{attribute addProperty BoxType "KL6224-0001"}
{attribute addProperty Id "Channel_1Channel_BED7D40000"}
{attribute addProperty CRC "1796210049"}
{attribute addProperty SizeInBites "0"}
{attribute addProperty SizeInBytes "0"}
TYPE KL_6B0FFD81 :
STRUCT
	{attribute addProperty Name "Channel_1"}
	Channel_1 : Channel_BED7D400;
END_STRUCT
END_TYPE

(* stored: Version 1.2.0.0, ProductVersion 3.1.4024.9
   DUT KL_6B0FFD81: Id {78bda593-89ce-4123-9093-2846120ab6f8} *)
